ABB RAPID module: MainModule.mod

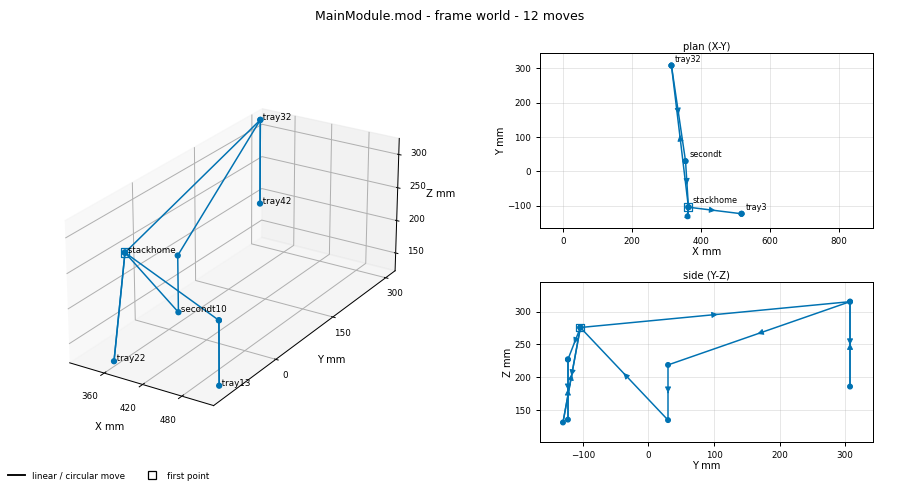
[picture p0: tool path of MainModule.mod in frame world, 12 of 12 moves have a stored position in this frame; points joined in program order, loops and branches not executed]
MODULE MainModule
	CONST robtarget p10:=[[295.05,-178.63,203.06],[0.705808,-0.037723,0.706379,-0.0379689],[-1,-1,-1,1],[9E+09,9E+09,9E+09,9E+09,9E+09,9E+09]];
	CONST robtarget p20:=[[358.45,-160.96,163.13],[0.705828,-0.0377255,0.706358,-0.0379887],[-1,-1,-1,1],[9E+09,9E+09,9E+09,9E+09,9E+09,9E+09]];
	CONST robtarget tray2:=[[365.66,-129.93,136.30],[0.719539,-0.053984,0.692332,0.00497193],[-1,-1,-1,1],[9E+09,9E+09,9E+09,9E+09,9E+09,9E+09]];
	CONST robtarget stackhome:=[[363.94,-103.75,275.83],[0.719395,-0.0539974,0.692481,0.00505825],[-1,-1,0,1],[9E+09,9E+09,9E+09,9E+09,9E+09,9E+09]];
	CONST robtarget tray22:=[[361.32,-130.30,130.99],[0.719418,-0.0540486,0.692453,0.00507747],[-1,-1,-1,1],[9E+09,9E+09,9E+09,9E+09,9E+09,9E+09]];
	CONST robtarget tray32:=[[314.62,307.51,315.25],[0.719409,-0.0540551,0.692461,0.00507583],[0,0,-1,1],[9E+09,9E+09,9E+09,9E+09,9E+09,9E+09]];
	CONST robtarget tray42:=[[314.62,307.51,185.75],[0.71942,-0.0540177,0.692453,0.00506861],[0,0,-1,1],[9E+09,9E+09,9E+09,9E+09,9E+09,9E+09]];
	CONST robtarget secondt:=[[355.56,29.95,218.77],[0.719338,-0.0540181,0.692538,0.00506612],[0,-1,-1,1],[9E+09,9E+09,9E+09,9E+09,9E+09,9E+09]];
	CONST robtarget secondt10:=[[355.55,29.95,134.59],[0.719319,-0.0540243,0.692557,0.00506541],[0,-1,-1,1],[9E+09,9E+09,9E+09,9E+09,9E+09,9E+09]];
	CONST robtarget stackhome10:=[[518.13,-122.75,227.14],[0.719245,-0.0541508,0.692624,0.00513783],[-1,-1,0,1],[9E+09,9E+09,9E+09,9E+09,9E+09,9E+09]];
	CONST robtarget tray3:=[[518.13,-122.75,227.14],[0.719245,-0.0541508,0.692624,0.00513783],[-1,-1,0,1],[9E+09,9E+09,9E+09,9E+09,9E+09,9E+09]];
	CONST robtarget tray13:=[[518.14,-122.75,135.34],[0.719259,-0.0541893,0.692606,0.00514018],[-1,-1,0,1],[9E+09,9E+09,9E+09,9E+09,9E+09,9E+09]];
	PROC main()
		MoveL stackhome, v100, z50, tool0;
		MoveL tray22, v100, z50, tool0;
		WaitTime 2;
		Set DO10_6;
		WaitTime 2;
		MoveL stackhome, v100, z50, tool0;
		MoveL tray32, v100, z50, tool0;
		MoveL tray42, v100, z50, tool0;
		WaitTime 2;
		Reset DO10_6;
		WaitTime 2;
		MoveL tray32, v100, z50, tool0;
		MoveL secondt, v100, z50, tool0;
		MoveL secondt10, v100, z50, tool0;
		WaitTime 2;
		Set DO10_6;
		WaitTime 2;
		MoveL stackhome, v100, z50, tool0;
		MoveL tray3, v100, z50, tool0;
		MoveL tray13, v100, z50, tool0;
		WaitTime 2;
		Set DO10_6;
		WaitTime 2;
		MoveL tray3, v100, z50, tool0;
	ENDPROC
ENDMODULE
